// TwinCAT 3 PLC project Plc
// ProgramVersion: 3.1.4024.0
// libraries:
//   Tc2_Standard, * (Beckhoff Automation GmbH)
//   Tc2_System, * (Beckhoff Automation GmbH)
//   Tc3_Module, * (Beckhoff Automation GmbH)
//   VisuDialogs, * (System)
// project tree:
//   / Gestore di visualizzazione.TcVMO (not stored), GlobalTextList.TcGTLO, ImagePool.TcIPO (not stored), PlcTask.TcTTO (not stored)
//   GVLs/ GVL.TcGVL
//   POUs/ MAIN.TcPOU
//   VISUs/ Visualization.TcVIS
// real-time tasks:
//   TASK PlcTask: cycle T#10ms, priority 20, ADS port 350
//   TASK VisuTask: cycle T#100000us, priority 60, ADS port 351

// ---- GVLs/GVL.TcGVL
{attribute 'qualified_only'}
VAR_GLOBAL
	//input
	PB1: BOOL; //Pulsante di start NA
	PB2: BOOL; //Pulsante di stop NC
	PBE: BOOL; //Pulsante di emergenza NC
	PS1: BOOL; //Fotocellula
	PS2: BOOL; //Fotocellula
	PS3: BOOL; //Fotocellula
	PS4: BOOL; //Fotocellula
	SB1: BOOL; //Finecorsa del sigillatore

	LS1: REAL; //Distanza misurata dal sensore laser [Volt]
	
	//output
	L1: BOOL; //Luce di segnalazione bianca
	L2: BOOL; //Luce di segnalazione verde
	L3: BOOL; //Luce di segnalazione blue
	L4: BOOL; //Luce di segnalazione gialla
	L5: BOOL; //Luce di segnalazione rossa
	M1 : BOOL; //Motore nastro 1
	M2 : BOOL; //Motore nastro 2

	P1 : BOOL; //Pistone sigillatore
	P2 : BOOL; //Pistone smistamento
END_VAR

// ---- POUs/MAIN.TcPOU
PROGRAM MAIN
VAR
	//Stati
	IN_FUNZIONE: BOOL;
	IN_SIGILLATURA: BOOL;
	IN_SMISTAMENTO: BOOL;
	SCATOLA_ALTA: BOOL;
	SCATOLA_BASSA: BOOL;
	
	//Timer
	TON_SIGILLATURA: TON;
	TON_RILEVAZIONE_ALTEZZA: TON;
	TON_SMISTAMENTO_ALTI: TON;

	//Counter
	CTU_ALTI: CTU;
	CTU_BASSI: CTU;
	STOP_CONFERMATO: BOOL;
	STOP_RICHIESTO: BOOL;
	TON_STOP: TON;
	IN_ANOMALIA: BOOL;
	TON_ANOMALIA: TON;
	CONTROLLO_ALTEZZA: BOOL;
	TON_ANOMALIA_ALTEZZA: TON;
	IN_RILEVAZIONE_ALTEZZA: BOOL;
	TON_FINECORSA_SIGILLATURA: TON;
	RILASCIA_PISTONE: BOOL;
END_VAR

GestioneAnomalie();
GestioneStop();
GestionePulsantiSegnalazioni();
GestioneMotori();
GestioneSigillatura();
GestioneSmistamento();
GestioneConteggio();

ACTION GestioneAnomalie:
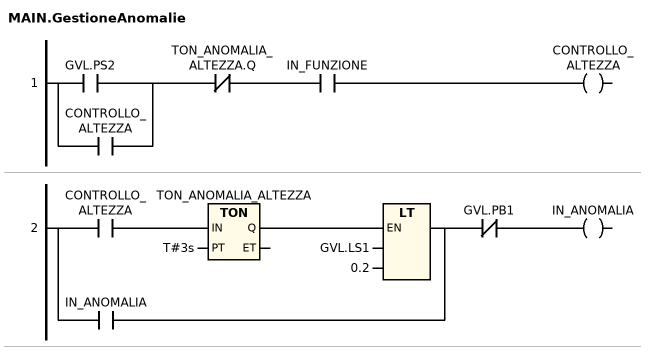
// NETWORK 1
CONTROLLO_ALTEZZA := (GVL.PS2 OR CONTROLLO_ALTEZZA) AND NOT TON_ANOMALIA_ALTEZZA.Q AND IN_FUNZIONE;

// NETWORK 2
TON_ANOMALIA_ALTEZZA(IN := CONTROLLO_ALTEZZA, PT := T#3s); // TON
IN_ANOMALIA := (TON_ANOMALIA_ALTEZZA.Q AND GVL.LS1 < 0.2 OR IN_ANOMALIA) AND NOT GVL.PB1;
END_ACTION

ACTION GestioneConteggio:
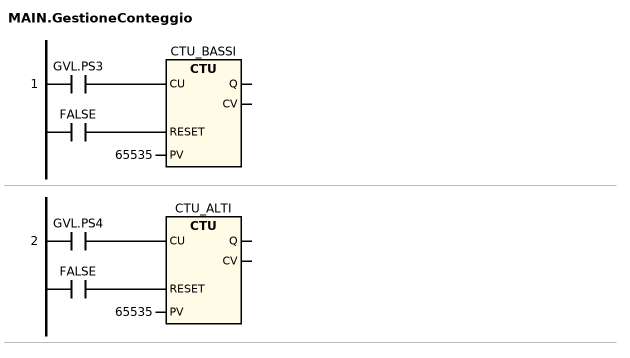
// NETWORK 1
CTU_BASSI(CU := GVL.PS3, RESET := FALSE, PV := 65535); // CTU

// NETWORK 2
CTU_ALTI(CU := GVL.PS4, RESET := FALSE, PV := 65535); // CTU
END_ACTION

ACTION GestioneMotori:
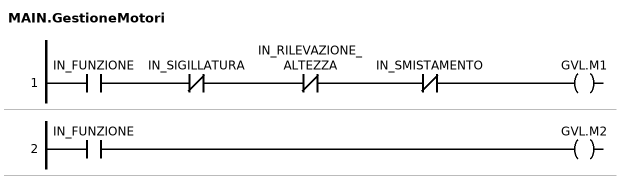
// NETWORK 1
GVL.M1 := IN_FUNZIONE AND NOT IN_SIGILLATURA AND NOT IN_RILEVAZIONE_ALTEZZA AND NOT IN_SMISTAMENTO;

// NETWORK 2
GVL.M2 := IN_FUNZIONE;
END_ACTION

ACTION GestionePulsantiSegnalazioni:
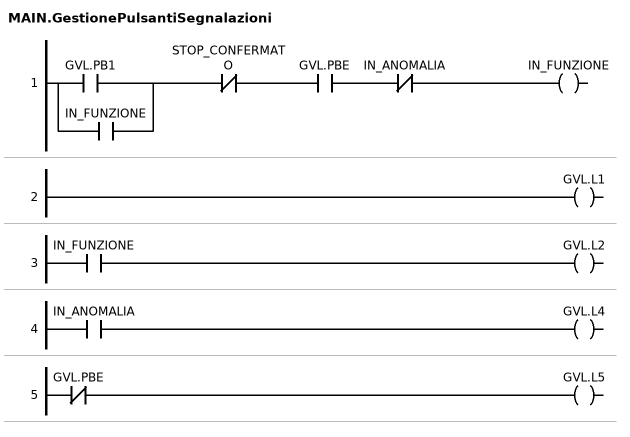
// NETWORK 1
IN_FUNZIONE := (GVL.PB1 OR IN_FUNZIONE) AND NOT STOP_CONFERMATO AND GVL.PBE AND NOT IN_ANOMALIA;

// NETWORK 2
GVL.L1 := TRUE;

// NETWORK 3
GVL.L2 := IN_FUNZIONE;

// NETWORK 4
GVL.L4 := IN_ANOMALIA;

// NETWORK 5
GVL.L5 := NOT GVL.PBE;
END_ACTION

ACTION GestioneSigillatura:
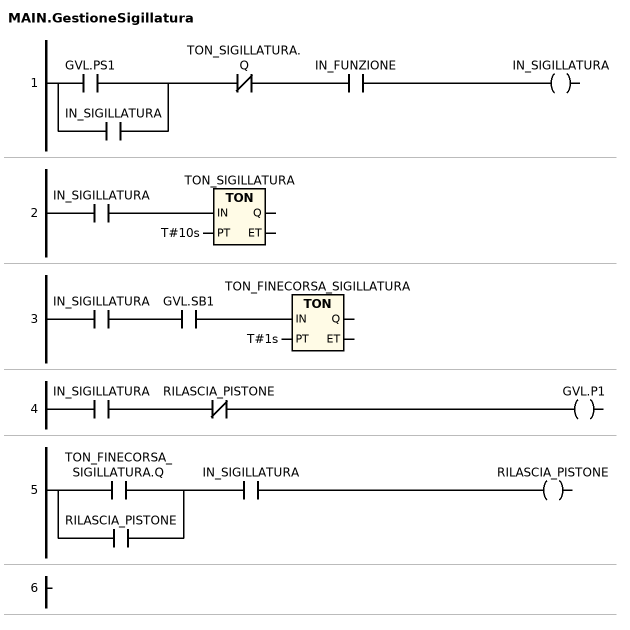
// NETWORK 1
IN_SIGILLATURA := (GVL.PS1 OR IN_SIGILLATURA) AND NOT TON_SIGILLATURA.Q AND IN_FUNZIONE;

// NETWORK 2
TON_SIGILLATURA(IN := IN_SIGILLATURA, PT := T#10s); // TON

// NETWORK 3
TON_FINECORSA_SIGILLATURA(IN := IN_SIGILLATURA AND GVL.SB1, PT := T#1s); // TON

// NETWORK 4
GVL.P1 := IN_SIGILLATURA AND NOT RILASCIA_PISTONE;

// NETWORK 5
RILASCIA_PISTONE := (TON_FINECORSA_SIGILLATURA.Q OR RILASCIA_PISTONE) AND IN_SIGILLATURA;

// NETWORK 6
END_ACTION

ACTION GestioneSmistamento:
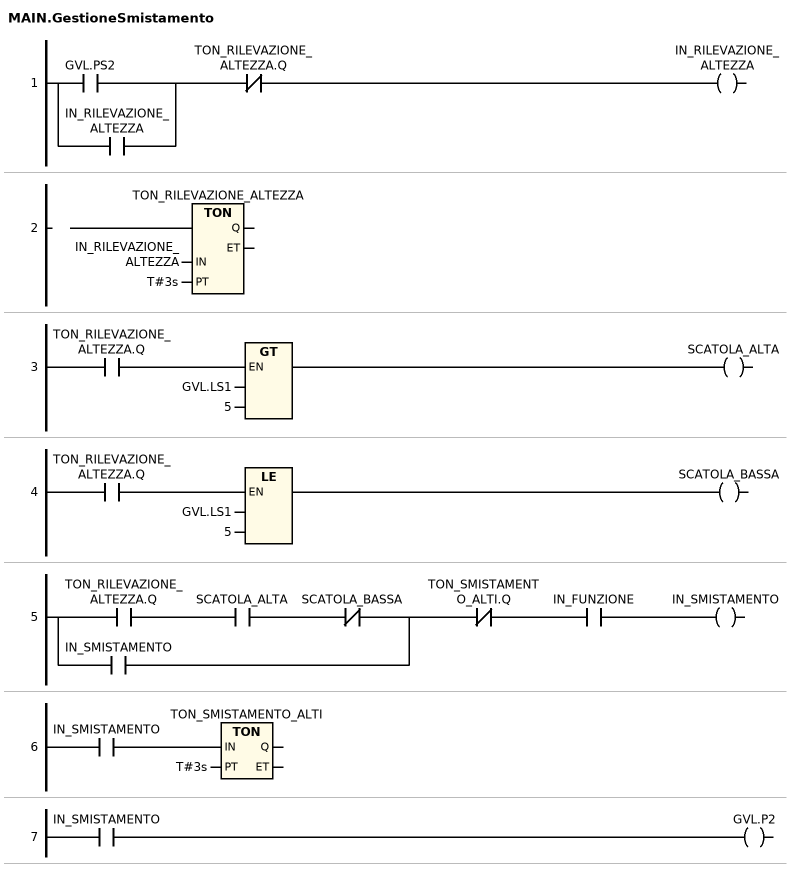
// NETWORK 1
IN_RILEVAZIONE_ALTEZZA := (GVL.PS2 OR IN_RILEVAZIONE_ALTEZZA) AND NOT TON_RILEVAZIONE_ALTEZZA.Q;

// NETWORK 2
TON_RILEVAZIONE_ALTEZZA(IN := IN_RILEVAZIONE_ALTEZZA, PT := T#3s); // TON

// NETWORK 3
SCATOLA_ALTA := TON_RILEVAZIONE_ALTEZZA.Q AND GVL.LS1 > 5;

// NETWORK 4
SCATOLA_BASSA := TON_RILEVAZIONE_ALTEZZA.Q AND GVL.LS1 <= 5;

// NETWORK 5
IN_SMISTAMENTO := (TON_RILEVAZIONE_ALTEZZA.Q AND SCATOLA_ALTA AND NOT SCATOLA_BASSA OR IN_SMISTAMENTO) AND NOT TON_SMISTAMENTO_ALTI.Q AND IN_FUNZIONE;

// NETWORK 6
TON_SMISTAMENTO_ALTI(IN := IN_SMISTAMENTO, PT := T#3s); // TON

// NETWORK 7
GVL.P2 := IN_SMISTAMENTO;
END_ACTION

ACTION GestioneStop:
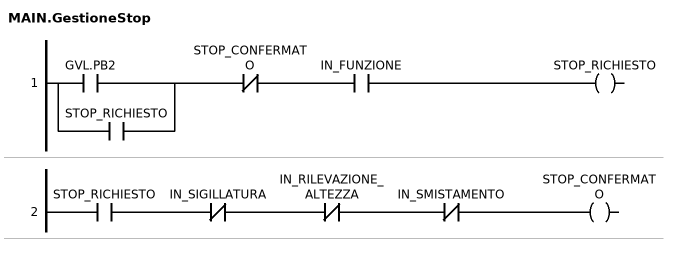
// NETWORK 1
STOP_RICHIESTO := (GVL.PB2 OR STOP_RICHIESTO) AND NOT STOP_CONFERMATO AND IN_FUNZIONE;

// NETWORK 2
STOP_CONFERMATO := STOP_RICHIESTO AND NOT IN_SIGILLATURA AND NOT IN_RILEVAZIONE_ALTEZZA AND NOT IN_SMISTAMENTO;
END_ACTION

END_PROGRAM

// ---- GlobalTextList.TcGTLO
TEXTLIST GlobalTextList
  628 = '%d'
  216 = '%f'
  108 = 'A11'
  331 = 'A12'
  600 = 'B11'
  978 = 'C'
  333 = 'C11'
  418 = 'contenitore'
  815 = 'contenitori'
  372 = 'CS_BIANCO'
  547 = 'CS_NERO'
  804 = 'Distanza [V]'
  68 = 'Emergenza'
  428 = 'EMERGENZA'
  304 = 'foratura'
  801 = 'FS1'
  524 = 'FS2'
  765 = 'LC1'
  869 = 'M1'
  802 = 'M2'
  115 = 'M3'
  287 = 'M4'
  498 = 'M5'
  465 = 'M_BLOCCO'
  962 = 'P1'
  268 = 'P2'
  35 = 'P3'
  951 = 'P4'
  324 = 'P5'
  501 = 'Percentuale prosciutti commerciabili: %d'
  820 = 'Percentuale prosciutti commerciabili:%d'
  57 = 'pistone'
  388 = 'PS1'
  310 = 'PS2'
  806 = 'PS3'
  525 = 'PS4'
  84 = 'PS5'
  843 = 'P_BLOCCO'
  656 = 'SB1'
  665 = 'SB2'
  112 = 'SB3'
  649 = 'Sensore Laser'
  881 = 'sigillatura'
  871 = 'Start'
  375 = 'START'
  275 = 'Stop'
  437 = 'STOP'
  800 = 'timbratura'
  305 = 'vasca di contenimento '
END_TEXTLIST

// ---- VISUs/Visualization.TcVIS
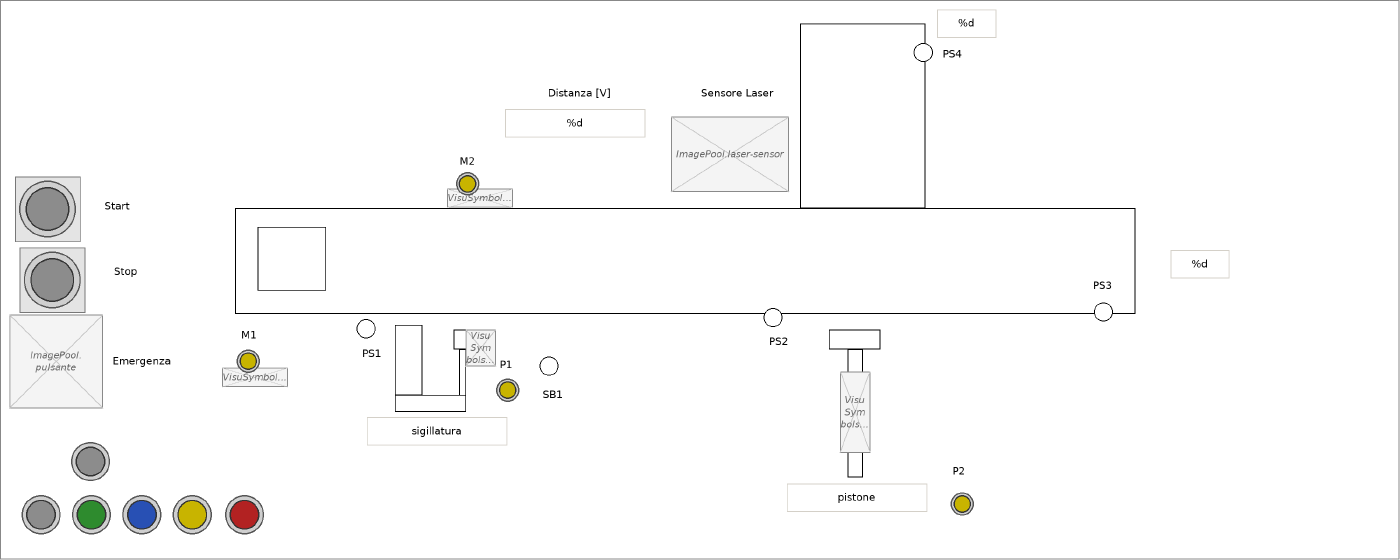
VISUALIZATION Visualization  // 1500x600
    RoundedRectangle (252,223 964x113)
    PushSwitch (16,189 70x70), variable: GVL.PB1, behaviour: TAP, style: Switch-PushSwitch-Gray
    Label (98,206 55x30), "Start"
    PushSwitch (21,265 70x70), variable: GVL.PB2, behaviour: TAP, style: Switch-PushSwitch-Gray
    Label (102,276 65x30), "Stop"
    Label (107,372 90x30), "Emergenza"
    Lamp1 (20,527 48x49), variable: GVL.L1, style: Lamp-Lamp1-Gray
    Lamp1 (74,527 48x49), variable: GVL.L2, style: Lamp-Lamp1-Green
    Lamp1 (128,527 48x49), variable: GVL.L3, style: Lamp-Lamp1-Blue
    Lamp1 (182,527 48x49), variable: GVL.L4, style: Lamp-Lamp1-Yellow
    Lamp1 (238,527 48x49), variable: GVL.L5, style: Lamp-Lamp1-Red
    Image (10,337 100x100), image: ImagePool.pulsante
        OnMouseClick: toggle GVL.PBE
    Textfield (843,518 150x30), "pistone"
    Rectangle (314,-68 198x134), angle 270
    RoundedRectangle (888,353 55x21)
    Rectangle (908,374 16x137)
    Image (900,398 32x87), image: VisuSymbols.Symbols.DoubleArrow4
    Rectangle (276,243 73x68)
    RoundedRectangle (486,353 19x21)
    Rectangle (492,374 7x51)
    Rectangle (423,423 76x18)
    Rectangle (423,348 29x75)
    Image (499,353 32x39), image: VisuSymbols.Symbols.DoubleArrow4
    Textfield (393,447 150x30), "sigillatura"
    Image (479,202 70x20), image: VisuSymbols.Symbols.ArrowBoldRight
    Image (238,394 70x20), image: VisuSymbols.Symbols.ArrowBoldRight
    Label (225,344 84x30), "M1"
    Label (459,158 84x30), "M2"
    Lamp1 (252,372 28x30), variable: GVL.M1, style: Lamp-Lamp1-Yellow
    Lamp1 (487,182 28x30), variable: GVL.M2, style: Lamp-Lamp1-Yellow
    Image (719,125 126x80), image: ImagePool.laser-sensor
    Lamp1 (1017,525 28x30), variable: GVL.P2, style: Lamp-Lamp1-Yellow
    Label (815,360 39x12), "PS2"
    Ellipse (818,330 20x20), colour toggle: GVL.PS2
        tap GVL.PS2
    Label (529,376 27x30), "P1"
    Lamp1 (530,403 28x30), variable: GVL.P1, style: Lamp-Lamp1-Yellow
    Ellipse (1172,324 20x20), colour toggle: GVL.PS3
        tap GVL.PS3
    Label (1162,300 39x12), "PS3"
    Textfield (1254,268 63x30), "%d", text variable: MAIN.CTU_BASSI.CV
    Lamp1 (73,470 48x49), variable: MAIN.STOP_RICHIESTO, style: Lamp-Lamp1-Gray
    Label (573,417 39x12), "SB1"
    Ellipse (578,382 20x20), colour toggle: GVL.SB1
        tap GVL.SB1
    Label (1014,490 27x30), "P2"
    Label (741,94 98x12), "Sensore Laser"
    Label (379,373 39x12), "PS1"
    Ellipse (382,342 20x20), colour toggle: GVL.PS1
        tap GVL.PS1
    Ellipse (979,46 20x20), colour toggle: GVL.PS4
        tap GVL.PS4
    Label (1001,52 39x12), "PS4"
    Textfield (1004,10 63x30), "%d", text variable: MAIN.CTU_ALTI.CV
    Textfield (541,117 150x30), "%d", text variable: GVL.LS1
        OnMouseClick: write the text variable via VisuDialogs.Numpad, min 0, max 10
    Label (572,94 98x12), "Distanza [V]"
END_VISUALIZATION
